# EPICS substitutions: iocBoot/ioc13ide/Pelco_CM6700.substitutions
file "$(IP)/ipApp/Db/Pelco_CM6700.db"
{
pattern
{P,       R,       PORT}
{13IDE:,  Pelco1,  serial7}
}

file "$(IP)/ipApp/Db/Pelco_CM6700_names.db"
{
pattern
{P,       R,       STR}
{13IDE:,  Pelco1,  ZRST}
{13IDE:,  Pelco1,  ONST}
{13IDE:,  Pelco1,  TWST}
{13IDE:,  Pelco1,  THST}
{13IDE:,  Pelco1,  FRST}
{13IDE:,  Pelco1,  FVST}
{13IDE:,  Pelco1,  SXST}
{13IDE:,  Pelco1,  SVST}
{13IDE:,  Pelco1,  EIST}
{13IDE:,  Pelco1,  NIST}
{13IDE:,  Pelco1,  TEST}
{13IDE:,  Pelco1,  ELST}
{13IDE:,  Pelco1,  TVST}
{13IDE:,  Pelco1,  TTST}
{13IDE:,  Pelco1,  FTST}
{13IDE:,  Pelco1,  FFST}
}
